FUNCTION WConcat6 : WSTRING(255)
VAR_INPUT
	wsExpression1: WSTRING(255);
	wsExpression2: WSTRING(255);
	wsExpression3: WSTRING(255);
	wsExpression4: WSTRING(255);
	wsExpression5: WSTRING(255);
	wsExpression6: WSTRING(255);
END_VAR

WConcat6 := WCONCAT(wsExpression1, wsExpression2);
WConcat6 := WCONCAT(WConcat6, wsExpression3);
WConcat6 := WCONCAT(WConcat6, wsExpression4);
WConcat6 := WCONCAT(WConcat6, wsExpression5);
WConcat6 := WCONCAT(WConcat6, wsExpression6);

END_FUNCTION

(* stored: Version 1.1.0.1, ProductVersion 3.1.4024.11
   POU WConcat6: Id {13d3f840-39e1-410f-863a-ef316af538bc}, SpecialFunc None *)
